FUNCTION_BLOCK FB_Door
VAR_INPUT
	tb_Enable_Doors														: BOOL;
	Open_Doors															: BOOL;
	Close_Doors															: BOOL;
	tb_Reset_doors															: BOOL;
	Open_Left_Door														: BOOL;
	Close_Left_Door														: BOOL;
	Open_Right_Door														: BOOL;
	Close_Right_Door													: BOOL;
	Left_Door_Closed_LS													: BOOL;
	Right_Door_Closed_LS												: BOOL;
	Left_Door_Open_LS													: BOOL;
	Right_Door_Open_LS													: BOOL;
	Left_Door_Clamps_Retracted											: BOOL;
	Right_Door_Clamps_Retracted											: BOOL;
	Max_Distance_To_Move												: REAL;
	Door_Position_Left													: REAL;
	Door_Position_Right													: REAL;
	Door_Ratio															: REAL;
	Door_Speed															: REAL	:= 4;
	Manual_Door_Position_Left											: REAL;
	Manual_Door_Position_Right											: REAL;
END_VAR

VAR_OUTPUT
	Enabled_Left														: BOOL;
	Enabled_Right														: BOOL;
	Homed_Left															: BOOL;
	Homed_Right															: BOOL;
	Moving_Left															: BOOL;
	Moving_Right														: BOOL;
	Current_Position_Left												: REAL;                           	
	Current_Position_Right												: REAL;                           	
	Done_Left															: BOOL;
	Done_Right															: BOOL;
	Error_Left															: STRING;
	Error_Right															: STRING;
END_VAR                             	
                             
VAR_IN_OUT
	Door_Axis_Left														: AXIS_REF;
	Door_Axis_Right														: AXIS_REF;
END_VAR
       	
VAR
	fbEnableLeft														: MC_Power;
	fbEnableRight														: MC_Power;
	fbResetLeft															: MC_Reset;
	fbResetRight														: MC_Reset;
	fbRunLeft															: MC_MoveRelative;
	fbRunRight															: MC_MoveRelative;
	fbMoveLeft															: MC_MoveAbsolute;
	fbMoveRight															: MC_MoveAbsolute;
	fbHomeLeft															: MC_Home;
	fbHomeRight															: MC_Home;
	fbHaltLeft															: MC_Halt;
	fbHaltRight															: MC_Halt;
	rtrigStart															: R_TRIG;
	rtrigClosedLeft														: R_TRIG;
	rtrigClosedRight													: R_TRIG;
	rtrigOpenLeft														: R_TRIG;
	rtrigOpenRight														: R_TRIG;
	sLeftError															: STRING; 
	sRightError															: STRING; 
	bReady																: BOOL;
	bOpen																: BOOL;
	bClose																: BOOL;
	bStartLeft															: BOOL;
	bStartRight															: BOOL;
	bMoveLeft															: BOOL;
	bMoveRight															: BOOL;
	bResetLeft															: BOOL;
	bResetRight															: BOOL;
	bLeftDoorPosChanged													: BOOL;
	bRightDoorPosChanged												: BOOL;
	rManual_Position_Left												: REAL;
	rManual_Position_Right												: REAL;
	rCurrent_Manual_Left_Pos											: REAL		:= -1;
	rCurrent_Manual_Right_Pos											: REAL		:= -1;
	rDistance															: REAL;
END_VAR

// FB_Door
// Rev 1.0 - February 6, 2024

Enabled_Left															:= (Door_Axis_Left.NcToPlc.StateDWord AND 2#00000001) = 0;	//1;
Enabled_Right															:= (Door_Axis_Right.NcToPlc.StateDWord AND 2#00000001) = 0;	//1;
Homed_Left																:= (Door_Axis_Left.NcToPlc.StateDWord AND 2#00000010) = 2;
Homed_Right																:= (Door_Axis_Right.NcToPlc.StateDWord AND 2#00000010) = 2;
Moving_Left																:= (Door_Axis_Left.NcToPlc.StateDWord AND 2#00000100) = 4;
Moving_Right															:= (Door_Axis_Right.NcToPlc.StateDWord AND 2#00000100) = 4;
Current_Position_Left													:= LREAL_TO_REAL(Door_Axis_Left.NcToPlc.ActPos) / Door_Ratio;
Current_Position_Right													:= LREAL_TO_REAL(Door_Axis_Right.NcToPlc.ActPos) / Door_Ratio;
Error_Left																:= SEL(sLeftError <> '', UDINT_TO_STRING(Door_Axis_Left.NcToPlc.ErrorCode), sLeftError);
Error_Right																:= SEL(sRightError <> '', UDINT_TO_STRING(Door_Axis_Right.NcToPlc.ErrorCode), sRightError);

IF tb_Reset_doors THEN
	bResetLeft															:= TRUE;
	bResetRight															:= TRUE;
END_IF

bReady																	:= Enabled_Left AND Enabled_Right AND NOT Moving_Left AND NOT Moving_Right;

IF Open_Doors THEN
	Open_Left_Door														:= TRUE;
	Open_Right_Door														:= TRUE;
	Open_Doors															:= FALSE;
ELSIF Close_Doors THEN
	Close_Left_Door														:= TRUE;
	Close_Right_Door													:= TRUE;
	Close_Doors															:= FALSE;
END_IF

bOpen																	:= Open_Left_Door OR Open_Right_Door;
bClose																	:= Close_Left_Door OR Close_Right_Door;
bLeftDoorPosChanged														:= Manual_Door_Position_Left <> -1 AND Manual_Door_Position_Left <> rCurrent_Manual_Left_Pos;
bRightDoorPosChanged													:= Manual_Door_Position_Right <> -1 AND Manual_Door_Position_Right <> rCurrent_Manual_Right_Pos;

rtrigStart(CLK:= (bOpen OR bClose OR bLeftDoorPosChanged OR bRightDoorPosChanged) AND bReady);

IF rtrigStart.Q THEN
	sLeftError															:= SEL((Open_Left_Door OR Close_Left_Door) AND NOT Left_Door_Clamps_Retracted, '', gsDoorClampsExtendedError);
	sRightError															:= SEL((Open_Right_Door OR Close_Right_Door) AND NOT Right_Door_Clamps_Retracted, '', gsDoorClampsExtendedError);
	IF sLeftError = '' AND sRightError = '' THEN
		IF bOpen OR bClose THEN
			rDistance													:= SEL(bOpen, 0 - Max_Distance_To_Move, Max_Distance_To_Move);
			bStartLeft													:= (Open_Left_Door AND NOT Left_Door_Open_LS) OR (Close_Left_Door AND NOT Left_Door_Closed_LS);
			bStartRight													:= (Open_Right_Door AND NOT Right_Door_Open_LS) OR (Close_Right_Door AND NOT Right_Door_Closed_LS);
			rCurrent_Manual_Left_Pos									:= -1;
			rCurrent_Manual_Right_Pos									:= -1;
		ELSE
			IF bLeftDoorPosChanged THEN
				rManual_Position_Left									:= Manual_Door_Position_Left;
				bMoveLeft												:= TRUE;
			END_IF
			IF bRightDoorPosChanged THEN
				rManual_Position_Right									:= Manual_Door_Position_Right;
				bMoveRight												:= TRUE;
			END_IF
		END_IF
	END_IF
ELSE
	bStartLeft															:= FALSE;
	bStartRight															:= FALSE;
	bMoveLeft															:= FALSE;
	bMoveRight															:= FALSE;
	Open_Left_Door														:= FALSE;
	Close_Left_Door														:= FALSE;
	Open_Right_Door														:= FALSE;
	Close_Right_Door													:= FALSE;
	sLeftError															:= '';
	sRightError															:= '';
END_IF
Manual_Door_Position_Left												:= -1;
Manual_Door_Position_Right												:= -1;

rtrigClosedLeft(CLK:= Left_Door_Closed_LS);
rtrigOpenLeft(CLK:= Left_Door_Open_LS);
rtrigClosedRight(CLK:= Right_Door_Closed_LS);
rtrigOpenRight(CLK:= Right_Door_Open_LS);

fbEnableLeft(	Axis													:= Door_Axis_Left,
				Enable													:= tb_Enable_Doors,
				Enable_Positive											:= TRUE, 
				Enable_Negative											:= TRUE, 
				Override												:= 100);
			                    				
fbEnableRight(	Axis													:= Door_Axis_Right,
				Enable													:= tb_Enable_Doors,
				Enable_Positive											:= TRUE, 
				Enable_Negative											:= TRUE, 
				Override												:= 100);
			                    				
fbResetLeft(	Axis													:= Door_Axis_Left,
				Execute													:= bResetLeft);
IF fbResetLeft.Error OR fbResetLeft.Done THEN
	Error_Left															:= SEL(fbResetLeft.ErrorID > 0, '', 'Left Reset Error');
	bResetLeft															:= FALSE;
END_IF

fbResetRight(	Axis													:= Door_Axis_Right,
				Execute													:= bResetRight);
IF fbResetRight.Error OR fbResetRight.Done THEN
	Error_Right															:= SEL(fbResetRight.ErrorID > 0, '', 'Right Reset Error');
	bResetRight															:= FALSE;
END_IF


fbRunLeft(		Axis													:= Door_Axis_Left, 
				Execute													:= bStartLeft, 
				Distance												:= rDistance, 
				Velocity												:= Door_Speed, 
				Done													=>, 
				Busy													=>, 
				Error													=> , 
				ErrorID													=> );
	                            	
fbRunRight(		Axis													:= Door_Axis_Right, 
				Execute													:= bStartRight, 
				Distance												:= rDistance, 
				Velocity												:= Door_Speed, 
				Done													=>, 
				Busy													=>, 
				Error													=> , 
				ErrorID													=> );

fbMoveLeft(		Axis													:= Door_Axis_Left,
				Execute													:= bMoveLeft, 
				Position												:= rManual_Position_Left, 
				Velocity												:= Door_Speed, 
				Acceleration											:= , 
				Deceleration											:= , 
				Jerk													:= , 
				Done													=> , 
				Busy													=> , 
				Active													=> , 
				CommandAborted											=> , 
				Error													=> , 
				ErrorID													=> );
IF fbMoveLeft.Done THEN
	rCurrent_Manual_Left_Pos											:= rManual_Position_Left;
END_IF
	                            	
fbMoveRight(	Axis													:= Door_Axis_Right,
				Execute													:= bMoveRight, 
				Position												:= rManual_Position_Right, 
				Velocity												:= Door_Speed, 
				Acceleration											:= , 
				Deceleration											:= , 
				Jerk													:= , 
				Done													=> , 
				Busy													=> , 
				Active													=> , 
				CommandAborted											=> , 
				Error													=> , 
				ErrorID													=> );
IF fbMoveRight.Done THEN
	rCurrent_Manual_Right_Pos											:= rManual_Position_Right;
END_IF
	                            	
fbHomeLeft(		Axis													:= Door_Axis_Left, 
				Execute													:= Left_Door_Closed_LS AND NOT Moving_Left,
				Position												:= 0, 
				HomingMode												:= MC_Direct,
				Done													=> );
			                    		
fbHomeRight(	Axis													:= Door_Axis_Right, 
				Execute													:= Right_Door_Closed_LS AND NOT Moving_Right,
				Position												:= 0, 
				HomingMode												:= MC_Direct,
				Done													=> );
			                    		
fbHaltLeft(		Axis													:= Door_Axis_Left, 
				Execute													:= Moving_Left AND (rtrigClosedLeft.Q OR rtrigOpenLeft.Q),
				Deceleration											:= DRIVE_STOP_DECEL, 
				Jerk													:= DRIVE_STOP_JERK,
				Done													=> Done_Left); 

fbHaltRight(	Axis													:= Door_Axis_Right, 
				Execute													:= Moving_Right AND (rtrigClosedRight.Q OR rtrigOpenRight.Q),
				Deceleration											:= DRIVE_STOP_DECEL, 
				Jerk													:= DRIVE_STOP_JERK,
				Done													=> Done_Right);

END_FUNCTION_BLOCK

(* stored: Version 1.1.0.1, ProductVersion 3.1.4024.12
   POU FB_Door: Id {4b0daecd-5988-4703-b41b-c2553a03edfd}, SpecialFunc None *)
